TYPE VFD :
STRUCT
	bStart : BOOL;
	bStop : BOOL;
	nRPMSetPointScaled : LREAL;
	nRPMFeedBackScaled : LREAL;
	nRPMFeedBackRaw : INT;
	nRPMSetPointRaw : INT;
END_STRUCT
END_TYPE

(* stored: Version 1.1.0.1, ProductVersion 3.1.4024.9
   DUT VFD: Id {f1541367-c265-476e-8313-219f1747d733} *)
